(* PLC project Unnamed, Неизвестно Unnamed 1 *)
(* stored: creationDateTime 2019-12-05T21:38:19, modificationDateTime 2019-12-11T19:39:32 *)

TYPE Mode_t : (inactive, started, holded, stopped) := inactive;
END_TYPE

FUNCTION calc_desired_tmp : REAL
  VAR_INPUT
    crnt_time : DINT;
    t1 : DINT;
    t2 : DINT;
    var1 : REAL;
    var2 : REAL;
  END_VAR

            calc_desired_tmp := var1 + (var2 - var1) * DINT_TO_REAL(crnt_time - t1) / DINT_TO_REAL(t2  - t1);
return;
          
END_FUNCTION

PROGRAM main
  VAR_EXTERNAL
    is_source_turned_on : BOOL;
    is_system_turned_on : BOOL;
    desired_first_temperature : REAL;
    desired_second_temperature : REAL;
    desired_first_holding : REAL;
    desired_second_holding : REAL;
    is_start_btn_pressed : BOOL;
    is_hold_btn_pressed : BOOL;
    is_stop_btn_pressed : BOOL;
    is_object_in_first_area : BOOL;
    is_object_between_areas : BOOL;
    is_object_in_second_area : BOOL;
    first_temperature : REAL;
    second_temperature : REAL;
    cmd_move_object : BOOL;
    mode : Mode_t;
    desired_first_current : REAL;
    desired_second_current : REAL;
    work_counter : DINT;
  END_VAR
  VAR
    delay_counter : DINT := 0;
  END_VAR
  VAR CONSTANT
    TASK_PERIOD_MS : INT := 20;
  END_VAR
  VAR
    FIRST_PERIOD_END_TICKS : INT;
    SECOND_PERIOD_END_TICKS : INT;
    THIRD_PERIOD_END_TICKS : INT;
    dummy_time : TIME := T#0D_0H_0M_0S_1MS;
    pid1 : PID;
    pid2 : PID;
  END_VAR
  VAR CONSTANT
    K_P : REAL := 0.001;
    K_I : REAL := 0.0001;
    K_D : REAL := 0.001;
  END_VAR
  VAR
    des1 : REAL;
    des2 : REAL;
    now1 : REAL;
    now2 : REAL;
  END_VAR

            (* 
@brief Define mode: process btn pressing
*)
if is_source_turned_on = true and is_system_turned_on = true then
  if is_start_btn_pressed = true then
    mode := started;
  elsif is_hold_btn_pressed = true then
    mode := holded;
  elsif is_stop_btn_pressed = true then
    mode := stopped;
  end_if;
else
  mode := inactive;
end_if;
is_start_btn_pressed := false;
is_hold_btn_pressed := false;
is_stop_btn_pressed := false;

(* Calculate desired control parameters in this moment *)
FIRST_PERIOD_END_TICKS := 10*(1000/TASK_PERIOD_MS) + DINT_TO_INT(delay_counter);
SECOND_PERIOD_END_TICKS := FIRST_PERIOD_END_TICKS + (REAL_TO_INT(desired_first_holding))*(1000/TASK_PERIOD_MS);
THIRD_PERIOD_END_TICKS := SECOND_PERIOD_END_TICKS + (REAL_TO_INT(desired_second_holding))*(1000/TASK_PERIOD_MS);

(* 
@brief Process timer
@note It uses to define which temperature should be used now.
*)
if mode = started then
  work_counter := work_counter + 1;
elsif mode = stopped or mode = inactive then
  work_counter := 0;
  delay_counter := 0;
end_if;

(* 
@brief Process object moving
@note Send command to move object and hold process while object is moving
*)
if work_counter < INT_TO_DINT(SECOND_PERIOD_END_TICKS) then
  cmd_move_object := false;
elsif work_counter = INT_TO_DINT(SECOND_PERIOD_END_TICKS) and is_object_in_first_area = true then
  cmd_move_object := true;
elsif work_counter = INT_TO_DINT(SECOND_PERIOD_END_TICKS) and is_object_in_second_area = true then
  cmd_move_object := false;
elsif work_counter = INT_TO_DINT(THIRD_PERIOD_END_TICKS) and is_object_in_second_area = true then
  cmd_move_object := true;
elsif work_counter = INT_TO_DINT(THIRD_PERIOD_END_TICKS) and is_object_in_second_area = false then
  cmd_move_object := false;
end_if;

if cmd_move_object = true then
  delay_counter := delay_counter + 1;
end_if;


(* 
@brief Set controlled data (desired first and second currents)
*)
now1 := first_temperature;
now2 := second_temperature;
if mode = started or mode = holded then
  (* 1. From 0 to 100 temperature *)
  if work_counter < INT_TO_DINT(FIRST_PERIOD_END_TICKS) and is_object_in_first_area = true then
    des1 := calc_desired_tmp(work_counter, 0, INT_TO_DINT(FIRST_PERIOD_END_TICKS), 24.0, 100.0);
    des2 := des1;
  (* 2. From 100 Ampers to first desired current *)
  elsif work_counter < INT_TO_DINT(SECOND_PERIOD_END_TICKS) and is_object_in_first_area = true then
    des1 := calc_desired_tmp(work_counter, INT_TO_DINT(FIRST_PERIOD_END_TICKS), INT_TO_DINT(SECOND_PERIOD_END_TICKS), 100.0, desired_first_temperature);
    des2 := des1;
  (* 3. Waiting while object between areas *)
  elsif (work_counter >= INT_TO_DINT(SECOND_PERIOD_END_TICKS)) and 
        (is_object_between_areas = true or is_object_in_first_area = true) then
    des1 := desired_first_temperature;
    des2 := desired_first_temperature;
  (* 4. From first desired temperature to second *)
  elsif work_counter < INT_TO_DINT(THIRD_PERIOD_END_TICKS) and is_object_in_second_area = true then
    des1 := desired_first_temperature;
    des2 := calc_desired_tmp(work_counter, INT_TO_DINT(SECOND_PERIOD_END_TICKS), INT_TO_DINT(THIRD_PERIOD_END_TICKS), desired_first_temperature, desired_second_temperature);
  else
    mode := stopped;
  end_if;
  pid1(true, des1, now1, 0.0, K_P, K_I, K_D, dummy_time, desired_first_current);
  pid2(true, des2, now2, 0.0, K_P, K_I, K_D, dummy_time, desired_second_current);
elsif mode = stopped then
  pid1(true, 24.0, now1, 0.0, K_P, K_I, K_D, dummy_time, desired_first_current);
  pid2(true, 24.0, now2, 0.0, K_P, K_I, K_D, dummy_time, desired_second_current);
end_if;
          
END_PROGRAM

PROGRAM simulation
  VAR_EXTERNAL
    is_source_turned_on : BOOL;
    is_system_turned_on : BOOL;
    is_reset_btn_pressed : BOOL;
    raw_first_current : INT;
    raw_second_current : INT;
    raw_first_temperature : INT;
    raw_second_temperature : INT;
    is_first_source_turned_on : BOOL;
    is_second_source_turned_on : BOOL;
    is_object_in_first_area : BOOL;
    is_object_between_areas : BOOL;
    is_object_in_second_area : BOOL;
    pwm_first_current : REAL;
    pwm_second_current : REAL;
    cmd_move_object : BOOL;
    MAX_CURRENT_VALUE : INT;
  END_VAR
  VAR
    real_temp_var : REAL;
  END_VAR
  VAR CONSTANT
    PWM_TO_TEMPERATURE : REAL := 40.0;
  END_VAR
  VAR_EXTERNAL
    work_counter : DINT;
  END_VAR
  VAR
    counter : INT := 0;
  END_VAR

            if is_source_turned_on = true then
  (* 1. Simulate currents *)
  real_temp_var := INT_TO_REAL(MAX_CURRENT_VALUE) * 0.01;
  raw_first_current := REAL_TO_INT(pwm_first_current * real_temp_var);
  raw_second_current := REAL_TO_INT(pwm_second_current * real_temp_var);
  
  (* 2. Simulate temperatures *)
  raw_first_temperature := 24 + REAL_TO_INT(PWM_TO_TEMPERATURE * pwm_first_current);
  raw_second_temperature := 24 + REAL_TO_INT(PWM_TO_TEMPERATURE * pwm_second_current);
  
  (* 3. Simulate object moving *)
  if cmd_move_object = true then
    counter := counter + 1;
    if counter > 275 then
      if is_object_in_first_area = true then
        is_object_in_first_area := false;
        is_object_between_areas := true;
      elsif is_object_between_areas = true then
        is_object_between_areas := false;
        is_object_in_second_area := true;
      elsif is_object_in_second_area = true then
        is_object_in_second_area := false;
        is_object_in_first_area := true;
      end_if;
      counter := 0;
    end_if;
  else
    counter := 0;
  end_if;

  if is_reset_btn_pressed = true then
    is_reset_btn_pressed := false;
    is_object_in_first_area := true;
    is_object_between_areas := false;
    is_object_in_second_area := false;
  end_if;
  
  
  (* 4. Make drift *)
  if mod(work_counter, 2) = 1 then
    raw_first_current := REAL_TO_INT(INT_TO_REAL(raw_first_current) * 1.01);
  elsif mod(work_counter, 3) = 1 then
    raw_first_current := REAL_TO_INT(INT_TO_REAL(raw_first_current) * 0.98);
  elsif mod(work_counter, 5) = 1 then
    raw_first_current := REAL_TO_INT(INT_TO_REAL(raw_first_current) * 1.03);
  elsif mod(work_counter, 7) = 1 then
    raw_first_current := REAL_TO_INT(INT_TO_REAL(raw_first_current) * 0.97);
  elsif mod(work_counter, 11) = 1 then
    raw_first_current := REAL_TO_INT(INT_TO_REAL(raw_first_current) * 1.04);
  end_if;
end_if;
          
END_PROGRAM

PROGRAM receive_signals
  VAR_EXTERNAL
    raw_first_current : INT;
    raw_second_current : INT;
    raw_first_temperature : INT;
    raw_second_temperature : INT;
    is_first_source_turned_on : BOOL;
    is_second_source_turned_on : BOOL;
    is_object_in_first_area : BOOL;
    is_object_between_areas : BOOL;
    is_object_in_second_area : BOOL;
    first_current : REAL;
    second_current : REAL;
    first_temperature : REAL;
    second_temperature : REAL;
  END_VAR

            (* 1. Parse current data *)
first_current := INT_TO_REAL(raw_first_current);
second_current := INT_TO_REAL(raw_second_current);

(* 2. Parse temperature data *)
first_temperature := INT_TO_REAL(raw_first_temperature);
second_temperature := INT_TO_REAL(raw_second_temperature);

(* 3. Parse object position *)
          
END_PROGRAM

PROGRAM transmite_signals
  VAR_EXTERNAL
    pwm_first_current : REAL;
    pwm_second_current : REAL;
    cmd_move_object : BOOL;
    cmd_enable_first_source : BOOL;
    cmd_enable_second_source : BOOL;
    desired_first_current : REAL;
    desired_second_current : REAL;
    MAX_CURRENT_VALUE : INT;
  END_VAR
  VAR
    real_temp_var : REAL;
  END_VAR

            real_temp_var := DIV(desired_first_current, INT_TO_REAL(MAX_CURRENT_VALUE));
pwm_first_current := real_temp_var * 100.0;

real_temp_var := DIV(desired_second_current, INT_TO_REAL(MAX_CURRENT_VALUE));
pwm_second_current := real_temp_var * 100.0;

(* Transmit move_object_cmd here*)

          
END_PROGRAM

CONFIGURATION config
  VAR_GLOBAL
    raw_first_current : INT;
    raw_second_current : INT;
    raw_first_temperature : INT;
    raw_second_temperature : INT;
    is_first_source_turned_on : BOOL;
    is_second_source_turned_on : BOOL;
    pwm_first_current : REAL;
    pwm_second_current : REAL;
    cmd_move_object : BOOL := 0;
    cmd_enable_first_source : BOOL;
    cmd_enable_second_source : BOOL;
    mode : Mode_t := stopped;
    desired_first_current : REAL := 0;
    desired_second_current : REAL := 0;
    work_counter : DINT := 0;
    MAX_CURRENT_VALUE : INT := 3000;
  END_VAR
  RESOURCE resource1 ON PLC
    TASK task0(INTERVAL := T#20ms, PRIORITY := 0);
    PROGRAM instance0 WITH task0 : main;
    PROGRAM instance2 WITH task0 : simulation;
    PROGRAM instance3 WITH task0 : receive_signals;
    PROGRAM instance4 WITH task0 : transmite_signals;
  END_RESOURCE
END_CONFIGURATION
